FUNCTION_BLOCK FB_PowderPip EXTENDS FB_GCodeTool

VAR

	//Specproperties
	pPneuChannelPress	: POINTER TO FB_PneuChannelRef;
	pPneuChannelVac		: POINTER TO FB_PneuChannelRef;
	
	nDOutChanValvePress	: USINT;	//Digitaler Ausgangskanal MzHead Druckventil
	nDOutChanValveVac	: USINT;	//Digitaler Ausgangskanal MzHead Vakuumventil 
	
	//****************************************Aktionvariablen****************************************************
	
	//Action: "InitTool"
	bInitTool			: BOOL;
	nStateA_InitTool	: USINT;	

	//Action: "SetPressure"
	bSetPress			: BOOL;
	fbSetPress			: FB_SetPressure;

	//Action: "SetVacuum"
	bSetVacuum			: BOOL;
	fbSetVacuum			: FB_SetPressure;
	
	//Action: "SwitchPressure"
	bSwitchPress		: BOOL;
	nStateA_SwitchPress	: USINT;	//State von A_SwitchPress()
	ePressCtrl			: E_PressCtrl;
	eCurrPressCtrl 		: E_PressCtrl; 
	tPressTime			: TIME;		//Öffnungszeit Druckventil
	timerPress			: TON;		//Timer für Öffnungszeit Druckventil
	
	//Action: "PulsePressure"
	bPulsePress			: BOOL;
	nStateA_PulsePress	: USINT;	//State von A_PulsePress()
	eSwitchCtrlPhase1	: E_PressCtrl;		//
	eSwitchCtrlPhase2	: E_PressCtrl;		//
	nPulseDutycycle		: UINT;		//Tastverhältnis (0-100%)
	nTimePhase1			: UINT;
	nTimePhase2			: UINT;
	timerPulse			: TON;		//Timer
	nSetpointPulses		: UINT;		//Soll Anzahl an Pulses
	nCurrentPulses		: UINT;		//aktuelle Anzahl an Pulses
	bPulseOn			: BOOL;	
	
	//Action: "PickPut
	bPickPut			: BOOL;
	nStateA_PickPut		: USINT;
	ePickPutMode		: E_PickPutMode;
	nIntakeVac			: INT;
	tIntakeTime			: TIME;
	nHoldVac			: INT;
	nBlowOutPress		: INT;
	nBlowOutPulseTime	: UINT;
	nBlowOutPulses		: UINT;
	timerPickPut		: TON;
	stActionDataPickPut	: ST_ActionData;	
	
END_VAR

IF eCurrentState = E_MachineState.MACHINESTATE_Active THEN
	
	IF bInitTool THEN
		A_InitTool();
		IF nStateA_InitTool >= 80 THEN
			IF nStateA_InitTool >= 99 THEN
				bError := TRUE;
			END_IF
			bInitTool := FALSE;
			nStateA_InitTool := 0;
			M_RemoveListEntry(nSearchValue:= E_Action.ACTION_Init);
		END_IF		
	END_IF
	
	IF bPickPut THEN
		A_PickPut();
		IF nStateA_PickPut >= 80 THEN
			IF nStateA_PickPut >= 99 THEN
				bError := TRUE;
			END_IF
			bPickPut := FALSE;
			nStateA_PickPut := 0;
			M_RemoveListEntry(nSearchValue:= E_Action.ACTION_PickPutPowder);
		END_IF
	END_IF		
	
	IF bSetPress THEN
		fbSetPress(pPneuChannelRef:= pPneuChannelPress);
		IF NOT fbSetPress.bBusy THEN
			IF fbSetPress.bError THEN
				bError := TRUE;
				stError.ErrorId := fbSetPress.nErrorId;
				stError.POU := E_POU.POU_FB_PowderPip;
				fbErrorList.M_Add(stError);
			END_IF
			bSetPress := FALSE;
			fbSetPress(pPneuChannelRef:= pPneuChannelPress, bExecute:= FALSE);
			M_RemoveListEntry(nSearchValue:= E_Action.ACTION_SetPressure);
		END_IF
	END_IF	

	IF bSetVacuum THEN
		fbSetVacuum(pPneuChannelRef:= pPneuChannelVac);
		IF NOT fbSetVacuum.bBusy THEN
			IF fbSetVacuum.bError THEN
				bError := TRUE;
				stError.ErrorId := fbSetVacuum.nErrorId;
				stError.POU := E_POU.POU_FB_PowderPip;
				fbErrorList.M_Add(stError);
			END_IF
			bSetVacuum := FALSE;
			fbSetVacuum(pPneuChannelRef:= pPneuChannelVac, bExecute:= FALSE);
			M_RemoveListEntry(nSearchValue:= E_Action.ACTION_SetVacuum);
		END_IF
	END_IF	

	IF bSwitchPress THEN	//Druck/Vakuum Ein/Aus
		A_SwitchPress();
		IF nStateA_SwitchPress >= 80 THEN
			IF nStateA_SwitchPress >= 99 THEN
				bError := TRUE;
			END_IF
			bSwitchPress := FALSE;
			nStateA_SwitchPress := 0;
			M_RemoveListEntry(nSearchValue:= E_Action.ACTION_SwitchPressure);
		END_IF
	END_IF
	
	IF bPulsePress THEN
		A_PulsePress();
		IF nStateA_PulsePress >= 80 THEN
			IF nStateA_PulsePress >= 99 THEN
				bError := TRUE;
			END_IF
			bPulsePress := FALSE;
			nStateA_PulsePress := 0;
			M_RemoveListEntry(nSearchValue:= E_Action.ACTION_PulsePressure);
		END_IF
	END_IF
END_IF

SUPER^();	//FB_MzTool aufrufen

//Prozessdaten aktualisieren

IF pPneuChannelPress > 0 THEN
	stProcessData.n32Data[7] := pPneuChannelPress^.P_nCurrentPressure;
	stProcessData.n32Data[8] := pPneuChannelPress^.P_nCurrentPressure;
END_IF

IF pPneuChannelVac > 0 THEN
	stProcessData.n32Data[9] := pPneuChannelVac^.P_nSetPressure;
	stProcessData.n32Data[10] := pPneuChannelVac^.P_nCurrentPressure;
END_IF

IF pZAxisRef > 0 THEN
	IF pZAxisRef^.stOutput.nToolCtrl = 0 THEN
		stProcessData.n32Data[11] := E_PressCtrl.PRESSCTRL_Off;
	ELSIF pZAxisRef^.stOutput.nToolCtrl = 5 THEN
		stProcessData.n32Data[11] := E_PressCtrl.PRESSCTRL_PressOn;
	ELSIF pZAxisRef^.stOutput.nToolCtrl = 3 THEN
		stProcessData.n32Data[11] := E_PressCtrl.PRESSCTRL_VacOn;
	ELSE
		stProcessData.n32Data[11] := E_PressCtrl.PRESSCTRL_UNDEFINED;
	END_IF
END_IF

aObjProcData[nNotifyId] := stProcessData;

ACTION A_InitTool:
IF nStateA_InitTool = 0 THEN
	IF nDOutChanValvePress > 0 THEN
		pFbMultiZ^.aDigiOut[nDOutChanValvePress] := TRUE;	
	END_IF
	IF nDOutChanValveVac > 0 THEN
		pFbMultiZ^.aDigiOut[nDOutChanValveVac] := TRUE;	
	END_IF
	bInitToolOk := TRUE;
	nStateA_InitTool := 80;
END_IF
END_ACTION

ACTION A_PickPut:
CASE nStateA_PickPut OF
	0:	//Ventile schließen
		pZAxisRef^.stOutput.nToolCtrl := 0;
		//Wenn Pick IntakeVac einstellen, bei Put BlowOutPress einstellen
		MEMSET(ADR(stActionDataPickPut),0,SIZEOF(stActionDataPickPut));
		IF ePickPutMode = E_PickPutMode.MODE_Pick THEN
			stActionDataPickPut.eAction := E_Action.ACTION_SetVacuum;
			stActionDataPickPut.aParams[2] := nIntakeVac;	
		ELSIF ePickPutMode = E_PickPutMode.MODE_Put THEN
			stActionDataPickPut.eAction := E_Action.ACTION_SetPressure;
			stActionDataPickPut.aParams[2] := nBlowOutPress;
			GVL_HwRefIO.bTrigger1 := TRUE;
		END_IF
		stActionDataPickPut.aParams[1] := 1;	//Fertigmeldung erst, wenn Druck erreicht
		stActionDataPickPut.aParams[3] := 8;	//Tolerance +
		stActionDataPickPut.aParams[4] := 8;	//Tolerance -
		stActionDataPickPut.aParams[5] := 10000; //Timeout
		M_ExeAction(stActionDataPickPut);
		stActionDataPickPut.eAction := E_Action.ACTION_SwitchPressure;
		stActionDataPickPut.aParams[1] := E_PressCtrl.PRESSCTRL_Off;
		M_ExeAction(stActionDataPickPut);
		nStateA_PickPut := 1;
	
	1:	//Warten bis SollDruck erreioht ist
		IF NOT M_GetActionBusy(E_Action.ACTION_SetPressure) AND NOT M_GetActionBusy(E_Action.ACTION_SetVacuum)THEN
			IF ePickPutMode = E_PickPutMode.MODE_Pick THEN
				nStateA_PickPut := 2;
			ELSE
				nStateA_PickPut := 20;
			END_IF
		END_IF
		
	2:	//Pick - Switch Vacuum
		MEMSET(ADR(stActionDataPickPut),0,SIZEOF(stActionDataPickPut));
		stActionDataPickPut.eAction := E_Action.ACTION_SwitchPressure;
		stActionDataPickPut.aParams[1] := E_PressCtrl.PRESSCTRL_VacOn;
		stActionDataPickPut.aParams[2] := 0;
		M_ExeAction(stActionDataPickPut);
		timerPickPut(IN:=TRUE, PT:= tIntakeTime);
		nStateA_PickPut := 3;

	3:	//Warten, bis Zeit abgelaufen
		timerPickPut();
		IF timerPickPut.Q THEN
			timerPickPut(IN:= FALSE);
			MEMSET(ADR(stActionDataPickPut),0,SIZEOF(stActionDataPickPut));
			//HoldVac einstellen (wenn HoldVac = 0, dann SwitchPress auf Off
			IF nHoldVac < 0 THEN
				stActionDataPickPut.eAction := E_Action.ACTION_SetVacuum;
				stActionDataPickPut.aParams[1] := 0; //Ohne Überwachung
				stActionDataPickPut.aParams[2] := nHoldVac;
				M_ExeAction(stActionDataPickPut);
			ELSE
				stActionDataPickPut.eAction := E_Action.ACTION_SwitchPressure;
				stActionDataPickPut.aParams[1] := E_PressCtrl.PRESSCTRL_Off;
				stActionDataPickPut.aParams[2] := 0;
				M_ExeAction(stActionDataPickPut);
			END_IF
			nStateA_PickPut := 80;
		END_IF
		
	20:	//Put
		//PulsePressure
		MEMSET(ADR(stActionDataPickPut),0,SIZEOF(stActionDataPickPut));
		stActionDataPickPut.eAction := E_Action.ACTION_PulsePressure;
		stActionDataPickPut.aParams[1] := E_PressCtrl.PRESSCTRL_PressOn;
		stActionDataPickPut.aParams[2] := E_PressCtrl.PRESSCTRL_Off;
		stActionDataPickPut.aParams[3] := nBlowOutPulseTime * 2; //Periode
		stActionDataPickPut.aParams[4] := 50; //Dutycycle
		stActionDataPickPut.aParams[5] := nBlowOutPulses;
		stActionDataPickPut.aParams[6] := 1; //On
		M_ExeAction(stActionDataPickPut);
		nStateA_PickPut := 21;
		
	21: //Warten, bis Pulsen fertig
		IF NOT M_GetActionBusy(E_Action.ACTION_PulsePressure) THEN
			GVL_HwRefIO.bTrigger1 := FALSE;
			nStateA_PickPut := 80;
		END_IF
	
	70: //Abbrechen
		M_CancelAction(E_Action.ACTION_PulsePressure);
		stActionDataPickPut.eAction := E_Action.ACTION_SwitchPressure;
		stActionDataPickPut.aParams[1] := E_PressCtrl.PRESSCTRL_Off;
		M_ExeAction(stActionDataPickPut);
		timerPickPut(IN:= FALSE);
		nStateA_PickPut := 80;
		
END_CASE
END_ACTION

ACTION A_PulsePress:
CASE nStateA_PulsePress OF
	0:	//Phase1
		
		IF eSwitchCtrlPhase1 = E_PressCtrl.PRESSCTRL_Off THEN
			pZAxisRef^.stOutput.nToolCtrl := 0;
		ELSIF eSwitchCtrlPhase1 = E_PressCtrl.PRESSCTRL_PressOn THEN
			pZAxisRef^.stOutput.nToolCtrl := 5;
		ELSIF eSwitchCtrlPhase1 = E_PressCtrl.PRESSCTRL_VacOn THEN
			pZAxisRef^.stOutput.nToolCtrl := 3;
		END_IF

		timerPulse(IN:= TRUE, PT:= UINT_TO_TIME(nTimePhase1));
		IF timerPulse.Q THEN
			timerPulse(IN:= FALSE);
			nStateA_PulsePress := 1;
			nCurrentPulses := nCurrentPulses + 1;
		END_IF

	1:	//Phase2

		IF eSwitchCtrlPhase2 = E_PressCtrl.PRESSCTRL_Off THEN
			pZAxisRef^.stOutput.nToolCtrl := 0;
		ELSIF eSwitchCtrlPhase2 = E_PressCtrl.PRESSCTRL_PressOn THEN
			pZAxisRef^.stOutput.nToolCtrl := 5;
		ELSIF eSwitchCtrlPhase2 = E_PressCtrl.PRESSCTRL_VacOn THEN
			pZAxisRef^.stOutput.nToolCtrl := 3;
		END_IF

		timerPulse(IN:= TRUE, PT:= UINT_TO_TIME(nTimePhase2));
		IF timerPulse.Q THEN
			timerPulse(IN:= FALSE);
			IF nCurrentPulses = nSetpointPulses THEN
				pZAxisRef^.stOutput.nToolCtrl := 0;
				nStateA_PulsePress := 80;
			ELSIF nSetpointPulses = 0 AND NOT bPulseOn THEN
				pZAxisRef^.stOutput.nToolCtrl := 0;
				nStateA_PulsePress := 80;
			ELSE
				nStateA_PulsePress := 0;	
			END_IF
		END_IF
		
	70:	//Abbrechen
		timerPulse(IN:= FALSE);
		pZAxisRef^.stOutput.nToolCtrl := 0;
		nStateA_PulsePress := 80;
		
END_CASE
END_ACTION

ACTION A_Reset:
//Ist noch eine Aktion aktiv?
IF nStateA_ResetSpec = 0 THEN 
	IF bSetPress THEN
		bSetPress := FALSE;
		fbSetPress(bExecute:= FALSE, pPneuChannelRef:= pPneuChannelPress);
	END_IF

	IF bSetVacuum THEN
		bSetVacuum := FALSE;
		fbSetVacuum(bExecute:= FALSE, pPneuChannelRef:= pPneuChannelVac);
	END_IF
	
	IF bSwitchPress THEN 
		bSwitchPress := FALSE;
		nStateA_SwitchPress := 0;
	END_IF
	
	IF bPulsePress THEN
		bPulsePress := FALSE;
		nStateA_PulsePress := 0;
	END_IF
	
	IF bPickPut THEN
		bPickPut := FALSE;
		nStateA_PickPut := 0;
	END_IF
	
	nStateA_ResetSpec := 80;
END_IF

SUPER^.A_Reset();
END_ACTION

ACTION A_Stop:
IF nStateA_Stop = 0 THEN

	IF bSetPress THEN
		fbSetPress(bExecute:= FALSE, pPneuChannelRef:= pPneuChannelPress);
	END_IF

	IF bSetVacuum THEN
		fbSetVacuum(bExecute:= FALSE, pPneuChannelRef:= pPneuChannelVac);
	END_IF

	IF bSwitchPress AND nStateA_SwitchPress < 70 THEN
		nStateA_SwitchPress := 70;
	END_IF
	
	IF bPulsePress AND nStateA_PulsePress < 70 THEN
		nStateA_PulsePress := 70;
	END_IF
	
	IF bPickPut AND nStateA_PickPut < 70 THEN
		nStateA_PickPut := 70;
	END_IF

	nStateA_Stop := 1;
END_IF

SUPER^.A_Stop();
END_ACTION

ACTION A_SwitchPress:
// In jedem Zustand sollte umgeschalten werden
CASE nStateA_SwitchPress OF
	0:	//Wie soll geschalten werden?
		IF ePressCtrl = E_PressCtrl.PRESSCTRL_Off THEN
			eCurrPressCtrl := E_PressCtrl.PRESSCTRL_Off;
			pZAxisRef^.stOutput.nToolCtrl := 0;
			timerPress(IN:= FALSE);
			nStateA_SwitchPress := 80;
			RETURN;
		ELSIF ePressCtrl = E_PressCtrl.PRESSCTRL_PressOn THEN
			eCurrPressCtrl := E_PressCtrl.PRESSCTRL_PressOn;
			pZAxisRef^.stOutput.nToolCtrl := 5;
		ELSIF ePressCtrl = E_PressCtrl.PRESSCTRL_VacOn THEN
			eCurrPressCtrl := E_PressCtrl.PRESSCTRL_VacOn;
			pZAxisRef^.stOutput.nToolCtrl := 3;
		END_IF

		IF tPressTime > T#0MS THEN
			timerPress(IN:= TRUE, PT:= tPressTime);
			nStateA_SwitchPress := 1;
		ELSE
			nStateA_SwitchPress := 80;
		END_IF
		
	1:	//Timer
		//Haben sich die Eingangsparameter geändert?
		IF ePressCtrl <> eCurrPressCtrl THEN
			nStateA_SwitchPress := 0;
			timerPress(IN:= FALSE);
		END_IF
		timerPress();
		IF timerPress.Q THEN
			timerPress(IN:= FALSE);
			pZAxisRef^.stOutput.nToolCtrl := 0;
			eCurrPressCtrl := E_PressCtrl.PRESSCTRL_Off;
			nStateA_SwitchPress := 80;
		END_IF

	70:	//Abbrechen
		pZAxisRef^.stOutput.nToolCtrl := 0;
		timerPress(IN:= FALSE);
		nStateA_SwitchPress := 80;
		
	80:	//Haben sich die Eingangsparameter geändert?
		IF ePressCtrl <> eCurrPressCtrl THEN
			nStateA_SwitchPress := 0;
		END_IF
END_CASE
END_ACTION

METHOD FB_init : BOOL
VAR_INPUT
	bInitRetains : BOOL; // if TRUE, the retain variables are initialized (warm start / cold start)
	bInCopyCode : BOOL;  // if TRUE, the instance afterwards gets moved into the copy code (online change)
END_VAR
eObjectType := E_ObjectType.OBJECTTYPE_PowderPip;
eObjectGroup := E_ObjectGroup.OBJECTGROUP_MzTool OR E_ObjectGroup.OBJECTGROUP_Device;
END_METHOD

METHOD M_AddChild : ERRORID
VAR_INPUT
	pObject : POINTER TO FB_Object;
	nSlotNr	: UINT;
	nIndex 	: INT;
END_VAR
//Kann folgende Objekt-Typen aufnehmen
//Nozzle
IF pObject > 0 THEN
	IF pObject^.P_eObjectType = E_ObjectType.OBJECTTYPE_Nozzle THEN
		M_AddChild := SUPER^.M_AddChild(pObject,nSlotNr,nIndex);
	ELSE
		M_AddChild := E_ErrorIdObjMgmt.ERRORID_InvalidParentObject;
	END_IF
ELSE
	M_AddChild := E_ErrorIdObjMgmt.ERRORID_InvalidParentObject;
END_IF
END_METHOD

METHOD M_CancelAction
VAR_INPUT
	eAction : E_Action;
END_VAR
CASE eAction OF
	E_Action.ACTION_SetPressure:
		IF bSetPress THEN
			fbSetPress(bExecute:= FALSE, pPneuChannelRef:= pPneuChannelPress);
		END_IF
	
	E_Action.ACTION_SetVacuum:
		IF bSetVacuum THEN
			fbSetVacuum(bExecute:= FALSE, pPneuChannelRef:= pPneuChannelVac);
		END_IF

	E_Action.ACTION_SwitchPressure:
		IF bSwitchPress AND nStateA_SwitchPress < 70 THEN
			nStateA_SwitchPress := 70;
		END_IF

	E_Action.ACTION_PickPutPowder:
		IF bPickPut AND nStateA_PickPut < 70 THEN
			nStateA_PickPut := 70;
		END_IF

	E_Action.ACTION_PulsePressure:
		IF bPulsePress AND nStateA_PulsePress < 70 THEN
			nStateA_PulsePress := 70;
		END_IF	
ELSE
	SUPER^.M_CancelAction(eAction);
END_CASE
END_METHOD

METHOD M_CheckAction : ERRORID
VAR_INPUT
	refActionData 	: REFERENCE TO ST_ActionData;
	pCorrelObject	: POINTER TO FB_Object;
END_VAR
IF refActionData.eAction = E_Action.ACTION_MeasureTool THEN
	IF fbObjectDirectory.M_GetObjType(refActionData.nTarget) <> E_ObjectType.OBJECTTYPE_TipCalibrator THEN
		M_CheckAction := E_ErrorIdCmd.ERRORID_UnsuitableTarget;
	END_IF
ELSE
	M_CheckAction := SUPER^.M_CheckAction(refActionData, pCorrelObject);
END_IF
END_METHOD

METHOD M_ExeAction : ERRORID
VAR_INPUT
	refActionData : REFERENCE TO ST_ActionData;	
END_VAR
IF NOT (eCurrentState = E_MachineState.MACHINESTATE_Idle OR
	eCurrentState = E_MachineState.MACHINESTATE_Active OR
	eCurrentState = E_MachineState.MACHINESTATE_Ready) THEN
	M_ExeAction := E_ErrorIdCmd.ERRORID_InvalidState;
	RETURN;
END_IF

CASE refActionData.eAction OF
	
	E_Action.ACTION_Init:
		IF NOT bInitAxis AND NOT bInitTool THEN
			bInitAxis := TRUE;
			bInitTool := TRUE;
			fbList.A_AddHeadValue( hList := hList, putValue := E_Action.ACTION_Init);	//InitBase
			fbList.A_AddHeadValue( hList := hList, putValue := E_Action.ACTION_Init);	//InitSpec
		ELSE
			RETURN;
		END_IF		

	E_Action.ACTION_SetPressure:
		fbSetPress(bExecute:= FALSE, pPneuChannelRef:= pPneuChannelPress); //eventueller Fehler wird auch zurückgesetzt
		fbSetPress.bAwait := DINT_TO_BOOL(refActionData.aParams[1]);
		fbSetPress.nValue := DINT_TO_INT(refActionData.aParams[2]);
		fbSetPress.nTolerancePlus := DINT_TO_INT(refActionData.aParams[3]);
		fbSetPress.nToleranceMinus := DINT_TO_INT(refActionData.aParams[4]);
		fbSetPress.tTimeout := DINT_TO_TIME(refActionData.aParams[5]);
		
		fbSetPress(bExecute:= TRUE,	pPneuChannelRef:= pPneuChannelPress,nErrorId=> M_ExeAction);
		IF fbSetPress.bError THEN
			RETURN;
		END_IF
		
		IF NOT bSetPress AND fbSetPress.bBusy THEN
			bSetPress := TRUE;
			fbList.A_AddHeadValue(hList := hList, putValue := E_Action.ACTION_SetPressure);
		ELSE
			RETURN;	
		END_IF

	E_Action.ACTION_SetVacuum:
		fbSetVacuum(bExecute:= FALSE, pPneuChannelRef:= pPneuChannelVac); //eventueller Fehler wird auch zurückgesetzt
		fbSetVacuum.bAwait := DINT_TO_BOOL(refActionData.aParams[1]);
		fbSetVacuum.nValue := DINT_TO_INT(refActionData.aParams[2]);
		fbSetVacuum.nTolerancePlus := DINT_TO_INT(refActionData.aParams[3]);
		fbSetVacuum.nToleranceMinus := DINT_TO_INT(refActionData.aParams[4]);
		fbSetVacuum.tTimeout := DINT_TO_TIME(refActionData.aParams[5]);
		
		fbSetVacuum(bExecute:= TRUE, pPneuChannelRef:= pPneuChannelVac,nErrorId=> M_ExeAction);
		IF fbSetVacuum.bError THEN
			RETURN;
		END_IF
		
		IF NOT bSetVacuum AND fbSetVacuum.bBusy THEN
			bSetVacuum := TRUE;
			fbList.A_AddHeadValue(hList := hList, putValue := E_Action.ACTION_SetVacuum);
		ELSE
			RETURN;	
		END_IF

	E_Action.ACTION_SwitchPressure:
		ePressCtrl := DINT_TO_USINT(refActionData.aParams[1]);
		tPressTime := DINT_TO_TIME(refActionData.aParams[2]);
		IF ePressCtrl = E_PressCtrl.PRESSCTRL_Off OR ePressCtrl = E_PressCtrl.PRESSCTRL_PressOn 
													OR ePressCtrl = E_PressCtrl.PRESSCTRL_VacOn THEN
			IF NOT bSwitchPress THEN
				fbList.A_AddHeadValue(hList := hList, putValue := E_Action.ACTION_SwitchPressure);
				bSwitchPress := TRUE;
			END_IF
		END_IF
				
	E_Action.ACTION_PulsePressure:
		bPulseOn := DINT_TO_BOOL(refActionData.aParams[6]);
		IF bPulseOn THEN	//On
			eSwitchCtrlPhase1 := DINT_TO_USINT(refActionData.aParams[1]);
			eSwitchCtrlPhase2 := DINT_TO_USINT(refActionData.aParams[2]);
	
			IF NOT(refActionData.aParams[4] >= 1 AND refActionData.aParams[4] <= 100) THEN
				M_ExeAction := E_ErrorIdCmd.ERRORID_InvalidDutyCycle;  //Error
				RETURN;
			END_IF
			nTimePhase1 := DINT_TO_UINT(refActionData.aParams[3] / 100 * refActionData.aParams[4]); 
			nTimePhase2 := DINT_TO_UINT(refActionData.aParams[3] - nTimePhase1);
			IF NOT bPulsePress THEN
				bPulsePress := TRUE;
				fbList.A_AddHeadValue(hList := hList, putValue := E_Action.ACTION_PulsePressure);
			ELSE
				RETURN;
			END_IF
			nCurrentPulses := 0;
			nSetpointPulses := DINT_TO_UINT(refActionData.aParams[5]);
		ELSE
			RETURN;
		END_IF				

	E_Action.ACTION_PickPutPowder:
		IF NOT bPickPut THEN
			ePickPutMode := DINT_TO_USINT(refActionData.aParams[1]);
			nIntakeVac := DINT_TO_INT(refActionData.aParams[2]);
			tIntakeTime := DINT_TO_TIME(refActionData.aParams[3]);
			nHoldVac := DINT_TO_INT(refActionData.aParams[4]);
			nBlowOutPress := DINT_TO_INT(refActionData.aParams[5]);
			nBlowOutPulseTime := DINT_TO_UINT(refActionData.aParams[6]);
			nBlowOutPulses := DINT_TO_UINT(refActionData.aParams[7]);
			IF nBlowOutPulseTime = 0 OR nBlowOutPulses = 0 THEN
				RETURN;
			END_IF
			bPickPut := TRUE;
			fbList.A_AddHeadValue(hList := hList, putValue := E_Action.ACTION_PickPutPowder);
		ELSE
			RETURN;	
		END_IF
	ELSE
		M_ExeAction := SUPER^.M_ExeAction(refActionData);
		RETURN;
END_CASE

bBusy := TRUE;
eCurrentState := E_MachineState.MACHINESTATE_Active;
END_METHOD

METHOD M_GetAllProps : ERRORID
VAR_INPUT
	refCmdData : REFERENCE TO  ST_CmdData;
END_VAR
//Basisproperties lesen
SUPER^.M_GetAllProps(refCmdData);
//Specialproperties lesen
nCurrentPropIndex := nCurrentPropIndex + 1; 
IF pPneuChannelPress > 0 THEN
	refCmdData.n32Data[nCurrentPropIndex] := pPneuChannelPress^.nChannel;
ELSE
	refCmdData.n32Data[nCurrentPropIndex] := 0;
END_IF

nCurrentPropIndex := nCurrentPropIndex + 1;
IF pPneuChannelVac > 0 THEN
	refCmdData.n32Data[nCurrentPropIndex] := pPneuChannelVac^.nChannel;
ELSE
	refCmdData.n32Data[nCurrentPropIndex] := 0;
END_IF

nCurrentPropIndex := nCurrentPropIndex + 1;
refCmdData.n32Data[nCurrentPropIndex] := nDOutChanValvePress; //Digitaler Ausgangskanal MzHead Druckventil
nCurrentPropIndex := nCurrentPropIndex + 1;
refCmdData.n32Data[nCurrentPropIndex] := nDOutChanValveVac;	//Digitaler Ausgangskanal MzHead Vakuumventil
END_METHOD

METHOD M_SetAllProps : ERRORID
VAR_INPUT
	refCmdData : REFERENCE TO  ST_CmdData;
END_VAR

VAR
	nPneuChannel : USINT;
END_VAR
M_SetAllProps := SUPER^.M_SetAllProps(refCmdData);

IF M_SetAllProps > 0 THEN
	RETURN;
END_IF

//PneuChannel Druck
nCurrentPropIndex := nCurrentPropIndex + 1;
nSpecPropIndex := nCurrentPropIndex;
nPneuChannel := DINT_TO_USINT(refCmdData.n32Data[nCurrentPropIndex]);
IF NOT (nPneuChannel > 0 AND nPneuChannel <= cNoOfPneuChannels) THEN
	M_SetAllProps := E_ErrorIdObjMgmt.ERRORID_InvalidPneuChannel;
	RETURN;	
END_IF
pPneuChannelPress := ADR(aFbPneuChannel[nPneuChannel]);

//PneuChannel Vakuum
nCurrentPropIndex := nCurrentPropIndex + 1;
nPneuChannel := DINT_TO_USINT(refCmdData.n32Data[nCurrentPropIndex]);		
IF NOT (nPneuChannel > 0 AND nPneuChannel <= cNoOfPneuChannels) THEN
	M_SetAllProps := E_ErrorIdObjMgmt.ERRORID_InvalidPneuChannel;
	RETURN;	
END_IF
pPneuChannelVac := ADR(aFbPneuChannel[nPneuChannel]);

nCurrentPropIndex := nCurrentPropIndex + 1;
nDOutChanValvePress := DINT_TO_USINT(refCmdData.n32Data[nCurrentPropIndex]); //Digitaler Ausgangskanal MzHead Druckventil Pressure
IF NOT(nDOutChanValvePress >= 0 AND nDOutChanValvePress <= 7) THEN
	M_SetAllProps := E_ErrorIdObjMgmt.ERRORID_InvalidMzDOutChannel;
	RETURN;
END_IF

nCurrentPropIndex := nCurrentPropIndex + 1;
nDOutChanValveVac := DINT_TO_USINT(refCmdData.n32Data[nCurrentPropIndex]);	//Digitaler Ausgangskanal MzHead Druckventil Vacuum
IF NOT(nDOutChanValveVac >= 0 AND nDOutChanValveVac <= 7) THEN	//kann 0 sein
	M_SetAllProps := E_ErrorIdObjMgmt.ERRORID_InvalidMzDOutChannel;
	RETURN;
END_IF

pZAxisRef^.eFixedToolType := E_MzToolType.TOOL_TYPE_PowderPip;

nNoOfProps := nCurrentPropIndex + 1;
END_METHOD

METHOD M_SetSingleProp : ERRORID
VAR_INPUT
	refCmdData : REFERENCE TO  ST_CmdData;
END_VAR

VAR
	nPneuChannel : USINT;
END_VAR
IF nSpecPropIndex = refCmdData.aHeader[1] THEN	//PneuChannel Druck
	nPneuChannel := DINT_TO_USINT(refCmdData.n32Data[0]);
	IF NOT (nPneuChannel > 0 AND nPneuChannel <= cNoOfPneuChannels) THEN
		M_SetSingleProp := E_ErrorIdObjMgmt.ERRORID_InvalidPneuChannel;
		RETURN;	
	END_IF
	pPneuChannelPress := ADR(aFbPneuChannel[nPneuChannel]);
ELSIF (nSpecPropIndex + 1) = refCmdData.aHeader[1] THEN //PneuChannel Vakuum
	nPneuChannel := DINT_TO_USINT(refCmdData.n32Data[0]);
	IF NOT (nPneuChannel >= 0 AND nPneuChannel <= cNoOfPneuChannels) THEN
		M_SetSingleProp := E_ErrorIdObjMgmt.ERRORID_InvalidPneuChannel;
		RETURN;	
	END_IF
	pPneuChannelVac := ADR(aFbPneuChannel[nPneuChannel]);		
ELSIF (nSpecPropIndex + 2) = refCmdData.aHeader[1] THEN //Digitaler Ausgangskanal MzHead Druckventil
	IF refCmdData.n32Data[0] < 1 OR refCmdData.n32Data[0] > 7 THEN	//Ausgang 1-7
		M_SetSingleProp := E_ErrorIdObjMgmt.ERRORID_InvalidMzDOutChannel;
		RETURN;
	END_IF
	nDOutChanValvePress := DINT_TO_USINT(refCmdData.n32Data[0]);	
ELSIF (nSpecPropIndex + 3) = refCmdData.aHeader[1] THEN //Digitaler Ausgangskanal MzHead Vakuumventil
	IF refCmdData.n32Data[0] < 1 OR refCmdData.n32Data[0] > 7 THEN	//Ausgang 1-7
		M_SetSingleProp := E_ErrorIdObjMgmt.ERRORID_InvalidMzDOutChannel;
		RETURN;
	END_IF
	nDOutChanValveVac := DINT_TO_USINT(refCmdData.n32Data[0]);	
ELSE
	M_SetSingleProp := SUPER^.M_SetSingleProp(refCmdData);
END_IF
END_METHOD

PROPERTY P_bIsInit : BOOL
GET
P_bIsInit := bInitToolOk AND SUPER^.P_bIsInit;
END_GET
END_PROPERTY

PROPERTY P_rToolRadius : REAL
GET
VAR
	stDim : ST_3DDimension;
END_VAR
P_rToolRadius := 4000.0;
END_GET
END_PROPERTY

END_FUNCTION_BLOCK

(* stored: Version 1.1.0.1, ProductVersion 3.1.4024.11
   POU FB_PowderPip: Id {920873ca-33ec-44ca-a287-8238e7a179ec}, SpecialFunc None
   Action A_InitTool: Id {e945e3c7-d464-4e65-9b41-dd2bae043b1a}
   Action A_PickPut: Id {cc0eb555-7174-4e3e-9775-e4388d127429}
   Action A_PulsePress: Id {48997c4d-c7be-4528-967c-7a3669245274}
   Action A_Reset: Id {790a71c5-b0cf-4782-8ec2-6e51c4c1da70}
   Action A_Stop: Id {35f6ee83-38fa-4c9b-914d-14c3c8088170}
   Action A_SwitchPress: Id {dee91c1c-fec1-45cf-b4d1-a7979a93f55f}
   Method FB_init: Id {f604e02c-8dfa-420c-a953-337f70c76b56}
   Method M_AddChild: Id {fd1483c6-4366-477b-a0ac-008d2b69db47}
   Method M_CancelAction: Id {5fe0de58-741f-43b6-90c3-abed53b7ea09}
   Method M_CheckAction: Id {8f3f8574-6368-4900-a58d-316d29c64d71}
   Method M_ExeAction: Id {26a823de-dab2-44ab-8669-325b727be060}
   Method M_GetAllProps: Id {e0cc6a9a-c37a-4e3a-8f9c-af193b5832c5}
   Method M_SetAllProps: Id {d16446ff-aeb9-4669-90b9-aaa00c76a71f}
   Method M_SetSingleProp: Id {2d022145-8ffa-4bcd-afa9-3f696dc0bd66}
   Property P_bIsInit: Id {3b4e5c0b-5709-4c7b-a5ca-136277dfbfec}
   Get Get: Id {b877ed27-4936-44b3-bda4-6b5047caad75}
   Property P_rToolRadius: Id {2c153cd9-73b9-46fd-8dd1-842697e9fabb}
   Get Get: Id {f95373ef-91f2-4fa4-b50b-914a5494358a} *)
